Fanuc KAREL source: kt00895.KL

-- PROVISIONAL review KL for V940-1; original PC SHA256 8356e87fb79a9d4469b7238626b5d10b80c36f622485c93729a089c31d36e578
-- Incomplete behavior may be omitted. Consult companion uncertainty JSON. Do not deploy.
PROGRAM KT00895
%NOLOCKGROUP
VAR
  OUT : BOOLEAN
-- UNRESOLVED_DECL P1 type=000106
-- UNRESOLVED_DECL P2 type=000106
BEGIN
  -- V9_ZERO_TABLE_METADATA_HINT layout=0001; no indexed target words; source/name/runtime held
  -- UNRESOLVED_PC offsets 5-20; opcodes 2E,22,32,35
  -- UNRESOLVED_PC offsets 25-40; opcodes 2E,22,32,35
  -- UNRESOLVED_PC offsets 45-60; opcodes 2E,22,32,35
  -- UNRESOLVED_PC offsets 65-80; opcodes 2E,22,32,35
  -- UNRESOLVED_PC offsets 85-108; opcodes 27,22,1C,27,9D,76,23
  -- UNRESOLVED_PC offsets 113-117; opcodes 7F
END KT00895
